FUNCTION_BLOCK ASSEMBLE_AL_FROM_AW (* this Function combines the 4 AW (WORD) adapters to a AL (LWORD) *)
  (* Standard: 61499-2; Description: Copyright (c) 2026 Meisterschulen am Ostbahnhof SPDX-License-Identifier: EPL-2.0 *)
  (* Version 1.0, 2026-05-16, Franz Höpfinger, Meisterschulen am Ostbahnhof, initial API and implementation and/or initial documentation *)
  PACKAGE adapter::assembling;
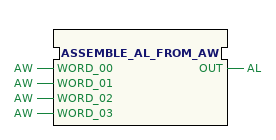
  SOCKETS
    WORD_00 : adapter::types::unidirectional::AW; (* Word 0 *)
    WORD_01 : adapter::types::unidirectional::AW; (* Word 1 *)
    WORD_02 : adapter::types::unidirectional::AW; (* Word 2 *)
    WORD_03 : adapter::types::unidirectional::AW; (* Word 3 *)
  END_SOCKETS
  PLUGS
    OUT : adapter::types::unidirectional::AL; (* LWORD Output *)
  END_PLUGS
END_FUNCTION_BLOCK
